// TIA Portal V20 export
TYPE "LKinCtrl_PathEditor_typePathTableInternalEvents"
// stored: Access Published
   STRUCT
      addChangeCommand { ExternalAccessible := 'False'; ExternalVisible := 'False'; ExternalWritable := 'False'} : Struct
         trigger : Bool;
         mode : USInt;   // 0: Add, 1:Edit
         programNo : DInt;
         commandNo : DInt;
         command : "LKinCtrl_typePathDataElement";
      END_STRUCT;
      updateTable { ExternalAccessible := 'False'; ExternalVisible := 'False'; ExternalWritable := 'False'} : Bool;
   END_STRUCT;
END_TYPE
